# EPICS StreamDevice protocol: waveStation3122App/Db/wavestation3122.proto
# streamDevice protocol file for WaveStation 3112

# @mismatch { disconnect; }
# @writetimeout { disconnect; }
# @readtimeout { disconnect; }
# @replyTimeout { disconnect; }

# OutTerminator = CR;
# InTerminator = CR;

# *IDN?
# IDN <device id>,<model>,<serial number>,<software version>,<firmware version>
# *IDN WST,WaveStation 3122,LCRY3601C00251,5.01.02.12,00-00-00-17-35\n

getIDN
{
    out "*IDN?";
    in  "*IDN WST,WaveStation 3122,%s\n";
    ExtraInput = Ignore;
}
